// TwinCAT 3 PLC project ReceipManager
// ProgramVersion: 3.1.4026.17
// libraries:
//   Tc2_Standard, * (Beckhoff Automation GmbH)
//   Tc2_System, * (Beckhoff Automation GmbH)
// project tree:
//   GVLs/ GVL_Command.TcGVL (not stored), GVL_Machine.TcGVL, GVL_Process.TcGVL, GVL_Recipe.TcGVL
//   / PlcTask.TcTTO
//   POUs/ FB_MachineSimulation.TcPOU, FB_ProcessStateMachine.TcPOU, MAIN.TcPOU

CONFIGURATION ReceipManager
    RESOURCE PLC ON TwinCAT3
        TASK PlcTask(INTERVAL := T#10ms, PRIORITY := 20);
        PROGRAM MAIN WITH PlcTask : MAIN;
    END_RESOURCE
END_CONFIGURATION

// ---- GVLs/GVL_Machine.TcGVL
{attribute 'qualified_only'}
VAR_GLOBAL
    MotorTemperature : REAL := 25.0;   // °C
    OilPressure : REAL := 3.0;         // bar
    MotorSpeed : REAL := 0.0;          // RPM

    TempWarning : BOOL := FALSE;
    PressureWarning : BOOL := FALSE;
    SpeedWarning : BOOL := FALSE;
END_VAR

// ---- GVLs/GVL_Process.TcGVL
{attribute 'qualified_only'}
VAR_GLOBAL
    CurrentStep : INT := 0;           // 0:Idle, 1..7 steps
    StepName : STRING(50) := 'Idle';

    Progress : REAL := 0.0;           // Global %
    StepProgress : REAL := 0.0;       // Step %
    
    StepTime_s : UDINT := 0;          // seconds in current step
    TotalTime_s : UDINT := 0;

    ErrorCode : INT := 0;
    ErrorText : STRING(100) := '';

    ProcessDone : BOOL := FALSE;
END_VAR

// ---- GVLs/GVL_Recipe.TcGVL
{attribute 'qualified_only'}
VAR_GLOBAL
    RecipeName : STRING(50) := '';
    NumIngredients : UDINT := 0;

    IngredientName : ARRAY[1..10] OF STRING(40);
    IngredientQuantity : ARRAY[1..10] OF REAL;     // en grammes
    IngredientVolume : ARRAY[1..10] OF REAL;       // en ml
    IngredientMolarMass : ARRAY[1..10] OF REAL;    // g/L
END_VAR

// ---- POUs/MAIN.TcPOU
PROGRAM MAIN
VAR
    fbProcess : FB_ProcessStateMachine;
    fbSim : FB_MachineSimulation;
    
    // Edge detection for start command
    StartEdge : R_TRIG;
END_VAR

// Simulation globale de la machine
fbSim();

// Detection du front montant de la commande Start
StartEdge(CLK := GVL_Command.StartProcess);

// Machine d'état du process
fbProcess(Start := StartEdge.Q);

// Fake ADS connection toggle for simulation
// In real application, this would be controlled by the ADS client
IF NOT GVL_Command.AdsConnected THEN
    GVL_Command.AdsConnected := TRUE;
END_IF

// Auto-reset process done flag after some time
// This allows running another process

END_PROGRAM

// ---- POUs/FB_ProcessStateMachine.TcPOU
FUNCTION_BLOCK FB_ProcessStateMachine
VAR_INPUT
    Start : BOOL;
END_VAR
VAR
    StepTimer : TON;
    RandomValue : DINT;
END_VAR

// Durée de chaque étape (Total: 30s)
VAR CONSTANT
    T_PREPARE : TIME := T#3s;
    T_DOSE_A : TIME := T#5s;
    T_DOSE_B : TIME := T#5s;
    T_MIX : TIME := T#10s;
    T_VERIFY : TIME := T#4s;
    T_FINALIZE : TIME := T#3s;
END_VAR

CASE GVL_Process.CurrentStep OF

    0: // Idle
        GVL_Process.StepName := 'Idle';
        GVL_Process.ProcessDone := FALSE;
        GVL_Process.Progress := 0.0;
        GVL_Process.StepProgress := 0.0;
        GVL_Process.StepTime_s := 0;
        
        IF Start THEN
            GVL_Process.CurrentStep := 1;
            GVL_Process.TotalTime_s := 0;
            GVL_Process.ErrorCode := 0;
            GVL_Process.ErrorText := '';
        END_IF

    1: // Preparation
        GVL_Process.StepName := 'Preparation';
        StepTimer(IN := TRUE, PT := T_PREPARE);

        GVL_Process.StepProgress := TIME_TO_REAL(StepTimer.ET) / TIME_TO_REAL(T_PREPARE);
        GVL_Process.Progress := GVL_Process.StepProgress * 0.1;
        GVL_Process.StepTime_s := TIME_TO_DINT(StepTimer.ET) / 1000;

        IF StepTimer.Q THEN
            StepTimer(IN := FALSE);
            GVL_Process.CurrentStep := 2;
        END_IF

    2: // Dose Ingredient A
        GVL_Process.StepName := 'Dosing Ingredient A';
        StepTimer(IN := TRUE, PT := T_DOSE_A);

        GVL_Process.StepProgress := TIME_TO_REAL(StepTimer.ET) / TIME_TO_REAL(T_DOSE_A);
        GVL_Process.Progress := 0.1 + GVL_Process.StepProgress * 0.2;
        GVL_Process.StepTime_s := TIME_TO_DINT(StepTimer.ET) / 1000;

        IF StepTimer.Q THEN
            StepTimer(IN := FALSE);
            GVL_Process.CurrentStep := 3;
        END_IF

    3: // Dose Ingredient B
        GVL_Process.StepName := 'Dosing Ingredient B';
        StepTimer(IN := TRUE, PT := T_DOSE_B);

        GVL_Process.StepProgress := TIME_TO_REAL(StepTimer.ET) / TIME_TO_REAL(T_DOSE_B);
        GVL_Process.Progress := 0.3 + GVL_Process.StepProgress * 0.2;
        GVL_Process.StepTime_s := TIME_TO_DINT(StepTimer.ET) / 1000;

        IF StepTimer.Q THEN
            StepTimer(IN := FALSE);
            GVL_Process.CurrentStep := 4;
        END_IF

    4: // Mixing
        GVL_Process.StepName := 'Mixing';
        StepTimer(IN := TRUE, PT := T_MIX);

        GVL_Process.StepProgress := TIME_TO_REAL(StepTimer.ET) / TIME_TO_REAL(T_MIX);
        GVL_Process.Progress := 0.5 + GVL_Process.StepProgress * 0.3;
        GVL_Process.StepTime_s := TIME_TO_DINT(StepTimer.ET) / 1000;

        IF StepTimer.Q THEN
            StepTimer(IN := FALSE);
            GVL_Process.CurrentStep := 5;
        END_IF

    5: // Verification
        GVL_Process.StepName := 'Verification';
        StepTimer(IN := TRUE, PT := T_VERIFY);

        GVL_Process.StepProgress := TIME_TO_REAL(StepTimer.ET) / TIME_TO_REAL(T_VERIFY);
        GVL_Process.Progress := 0.8 + GVL_Process.StepProgress * 0.1;
        GVL_Process.StepTime_s := TIME_TO_DINT(StepTimer.ET) / 1000;

        IF StepTimer.Q THEN
            StepTimer(IN := FALSE);
            GVL_Process.CurrentStep := 6;
        END_IF

    6: // Finalizing
        GVL_Process.StepName := 'Finalizing';
        StepTimer(IN := TRUE, PT := T_FINALIZE);

        GVL_Process.StepProgress := TIME_TO_REAL(StepTimer.ET) / TIME_TO_REAL(T_FINALIZE);
        GVL_Process.Progress := 0.9 + GVL_Process.StepProgress * 0.1;
        GVL_Process.StepTime_s := TIME_TO_DINT(StepTimer.ET) / 1000;

        IF StepTimer.Q THEN
            StepTimer(IN := FALSE);
            GVL_Process.CurrentStep := 7;
        END_IF

    7: // Done
        GVL_Process.StepName := 'Done';
        GVL_Process.Progress := 1.0;
        GVL_Process.ProcessDone := TRUE;
        GVL_Process.StepProgress := 1.0;
        
        // Reset to idle after some time or manual reset
        IF GVL_Command.ResetProcess THEN
            GVL_Process.CurrentStep := 0;
        END_IF
END_CASE

// Update total time
IF GVL_Process.CurrentStep > 0 AND GVL_Process.CurrentStep < 7 THEN
    GVL_Process.TotalTime_s := GVL_Process.TotalTime_s + 1;
END_IF

END_FUNCTION_BLOCK

// ---- POUs/FB_MachineSimulation.TcPOU
FUNCTION_BLOCK FB_MachineSimulation
VAR
    RandomSeed : DINT := 12345;
    Counter : UDINT := 0;
    TargetTemp : REAL := 25.0;
    TargetPressure : REAL := 1.0;
    TargetSpeed : REAL := 0.0;
END_VAR

Counter := Counter + 1;

// Simple random simulation
RandomSeed := (RandomSeed * 1103515245 + 12345) MOD 2147483647;

// Set target values based on current process step (pharmaceutical process simulation)
CASE GVL_Process.CurrentStep OF
    0: // Idle
        TargetTemp := 25.0;
        TargetPressure := 1.0;
        TargetSpeed := 0.0;
        
    1: // Preparation
        TargetTemp := 25.0;
        TargetPressure := 1.0;
        TargetSpeed := 0.0;
        
    2: // Dosing Ingredient A
        TargetTemp := 30.0;
        TargetPressure := 1.0;
        TargetSpeed := 150.0;
        
    3: // Dosing Ingredient B
        TargetTemp := 45.0;
        TargetPressure := 1.2;
        TargetSpeed := 200.0;
        
    4: // Mixing
        TargetTemp := 85.0;
        TargetPressure := 1.5;
        TargetSpeed := 350.0;
        
    5: // Verification/Cooling
        TargetTemp := 40.0;
        TargetPressure := 1.2;
        TargetSpeed := 200.0;
        
    6: // Finalizing
        TargetTemp := 25.0;
        TargetPressure := 1.0;
        TargetSpeed := 0.0;
        
    7: // Done
        TargetTemp := 25.0;
        TargetPressure := 1.0;
        TargetSpeed := 0.0;
END_CASE

// Simulate machine behavior with gradual transitions to target values
IF GVL_Process.CurrentStep > 0 AND GVL_Process.CurrentStep < 7 THEN
    // Gradually adjust temperature towards target
    IF ABS(GVL_Machine.MotorTemperature - TargetTemp) > 0.5 THEN
        IF GVL_Machine.MotorTemperature < TargetTemp THEN
            GVL_Machine.MotorTemperature := GVL_Machine.MotorTemperature + 0.2;
        ELSE
            GVL_Machine.MotorTemperature := GVL_Machine.MotorTemperature - 0.2;
        END_IF
    ELSE
        GVL_Machine.MotorTemperature := TargetTemp;
    END_IF
    
    // Add small random fluctuations to temperature
    GVL_Machine.MotorTemperature := GVL_Machine.MotorTemperature + (DINT_TO_REAL(RandomSeed MOD 20) - 10.0) / 20.0;
    
    // Gradually adjust speed towards target
    IF ABS(GVL_Machine.MotorSpeed - TargetSpeed) > 5.0 THEN
        IF GVL_Machine.MotorSpeed < TargetSpeed THEN
            GVL_Machine.MotorSpeed := GVL_Machine.MotorSpeed + 5.0;
        ELSE
            GVL_Machine.MotorSpeed := GVL_Machine.MotorSpeed - 5.0;
        END_IF
    ELSE
        GVL_Machine.MotorSpeed := TargetSpeed;
    END_IF
    
    // Add small random fluctuations to speed
    IF TargetSpeed > 0.0 THEN
        GVL_Machine.MotorSpeed := GVL_Machine.MotorSpeed + (DINT_TO_REAL(RandomSeed MOD 10) - 5.0);
    END_IF
    
    // Gradually adjust pressure towards target
    IF ABS(GVL_Machine.OilPressure - TargetPressure) > 0.05 THEN
        IF GVL_Machine.OilPressure < TargetPressure THEN
            GVL_Machine.OilPressure := GVL_Machine.OilPressure + 0.02;
        ELSE
            GVL_Machine.OilPressure := GVL_Machine.OilPressure - 0.02;
        END_IF
    ELSE
        GVL_Machine.OilPressure := TargetPressure;
    END_IF
    
    // Add small random fluctuations to pressure
    GVL_Machine.OilPressure := GVL_Machine.OilPressure + (DINT_TO_REAL(RandomSeed MOD 10) - 5.0) / 100.0;
    
ELSIF GVL_Process.CurrentStep = 0 THEN
    // Idle state
    GVL_Machine.MotorSpeed := 0.0;
    
    // Temperature cools down to ambient
    IF GVL_Machine.MotorTemperature > 25.0 THEN
        GVL_Machine.MotorTemperature := GVL_Machine.MotorTemperature - 0.1;
    ELSIF GVL_Machine.MotorTemperature < 25.0 THEN
        GVL_Machine.MotorTemperature := GVL_Machine.MotorTemperature + 0.1;
    END_IF
    
    // Pressure returns to atmospheric
    IF GVL_Machine.OilPressure > 1.0 THEN
        GVL_Machine.OilPressure := GVL_Machine.OilPressure - 0.02;
    ELSIF GVL_Machine.OilPressure < 1.0 THEN
        GVL_Machine.OilPressure := GVL_Machine.OilPressure + 0.02;
    END_IF
    
ELSE
    // Done state
    GVL_Machine.MotorSpeed := 0.0;
    
    // Maintain final temperature
    IF GVL_Machine.MotorTemperature > 25.0 THEN
        GVL_Machine.MotorTemperature := GVL_Machine.MotorTemperature - 0.05;
    END_IF
    
    GVL_Machine.OilPressure := 1.0;
END_IF

// Warning flags based on pharmaceutical process limits
GVL_Machine.TempWarning := (GVL_Machine.MotorTemperature > 95.0) OR (GVL_Machine.MotorTemperature < 15.0);
GVL_Machine.PressureWarning := (GVL_Machine.OilPressure < 0.5) OR (GVL_Machine.OilPressure > 2.0);
GVL_Machine.SpeedWarning := (GVL_Machine.MotorSpeed > 400.0);

// Simulate random anomaly (0.5% chance per cycle, reduced from 1%)
IF (RandomSeed MOD 200) = 0 AND GVL_Process.CurrentStep > 0 AND GVL_Process.CurrentStep < 7 THEN
    GVL_Process.ErrorCode := 1;
    GVL_Process.ErrorText := 'Sensor anomaly detected';
END_IF

END_FUNCTION_BLOCK
